FUNCTION_BLOCK FB_LensCompounder_Test EXTENDS TcUnit.FB_TestSuite
VAR
    nTestID : INT;
END_VAR


nTestID := 0;

Test0FocalLengthExpectError0FocalLength();

Test0MultiplierExpectError0FocalLength();

TestNegMultiplierExpectError0FocalLength();

TestResetExpectNoErrorAccurateFocalLength();

TestResetExpectNoErrorAccurateFocalLength_1();

// Expected results taken from pcdscalc/be_lens_calcs.py.
// Element = Be. Test Count = 1.
TestValidInputsExpectNoErrorAccurateFocalLength(
    fFocalLength1 := 0.008893754309452119,
    nMultiplier1 := 1,
    fFocalLength2 := 0.008893754309452119,
    nMultiplier2 := 1,
    fExpected := 0.004446877154726059
);

// Expected results taken from pcdscalc/be_lens_calcs.py.
// Element = Be. Test Count = 2.
TestValidInputsExpectNoErrorAccurateFocalLength(
    fFocalLength1 := 0.008893754309452119,
    nMultiplier1 := 1,
    fFocalLength2 := 0.008893754309452119,
    nMultiplier2 := 2,
    fExpected := 0.002964584769817373
);

// Expected results taken from pcdscalc/be_lens_calcs.py.
// Element = Be. Test Count = 3.
TestValidInputsExpectNoErrorAccurateFocalLength(
    fFocalLength1 := 0.008893754309452119,
    nMultiplier1 := 2,
    fFocalLength2 := 0.008893754309452119,
    nMultiplier2 := 1,
    fExpected := 0.002964584769817373
);

// Expected results taken from pcdscalc/be_lens_calcs.py.
// Element = Be. Test Count = 4.
TestValidInputsExpectNoErrorAccurateFocalLength(
    fFocalLength1 := 0.008893754309452119,
    nMultiplier1 := 2,
    fFocalLength2 := 0.008893754309452119,
    nMultiplier2 := 2,
    fExpected := 0.0022234385773630297
);

// Expected results taken from pcdscalc/be_lens_calcs.py.
// Element = Be. Test Count = 5.
TestValidInputsExpectNoErrorAccurateFocalLength(
    fFocalLength1 := 0.008893754309452119,
    nMultiplier1 := 1,
    fFocalLength2 := 0.45358146978205804,
    nMultiplier2 := 1,
    fExpected := 0.008722720572731886
);

// Expected results taken from pcdscalc/be_lens_calcs.py.
// Element = Be. Test Count = 6.
TestValidInputsExpectNoErrorAccurateFocalLength(
    fFocalLength1 := 0.008893754309452119,
    nMultiplier1 := 1,
    fFocalLength2 := 0.45358146978205804,
    nMultiplier2 := 2,
    fExpected := 0.008558140939284115
);

// Expected results taken from pcdscalc/be_lens_calcs.py.
// Element = Be. Test Count = 7.
TestValidInputsExpectNoErrorAccurateFocalLength(
    fFocalLength1 := 0.008893754309452119,
    nMultiplier1 := 2,
    fFocalLength2 := 0.45358146978205804,
    nMultiplier2 := 1,
    fExpected := 0.004403703590117068
);

// Expected results taken from pcdscalc/be_lens_calcs.py.
// Element = Be. Test Count = 8.
TestValidInputsExpectNoErrorAccurateFocalLength(
    fFocalLength1 := 0.008893754309452119,
    nMultiplier1 := 2,
    fFocalLength2 := 0.45358146978205804,
    nMultiplier2 := 2,
    fExpected := 0.004361360286365943
);

// Expected results taken from pcdscalc/be_lens_calcs.py.
// Element = Be. Test Count = 9.
TestValidInputsExpectNoErrorAccurateFocalLength(
    fFocalLength1 := 0.45358146978205804,
    nMultiplier1 := 1,
    fFocalLength2 := 0.008893754309452119,
    nMultiplier2 := 1,
    fExpected := 0.008722720572731886
);

// Expected results taken from pcdscalc/be_lens_calcs.py.
// Element = Be. Test Count = 10.
TestValidInputsExpectNoErrorAccurateFocalLength(
    fFocalLength1 := 0.45358146978205804,
    nMultiplier1 := 1,
    fFocalLength2 := 0.008893754309452119,
    nMultiplier2 := 2,
    fExpected := 0.004403703590117068
);

// Expected results taken from pcdscalc/be_lens_calcs.py.
// Element = Be. Test Count = 11.
TestValidInputsExpectNoErrorAccurateFocalLength(
    fFocalLength1 := 0.45358146978205804,
    nMultiplier1 := 2,
    fFocalLength2 := 0.008893754309452119,
    nMultiplier2 := 1,
    fExpected := 0.008558140939284115
);

// Expected results taken from pcdscalc/be_lens_calcs.py.
// Element = Be. Test Count = 12.
TestValidInputsExpectNoErrorAccurateFocalLength(
    fFocalLength1 := 0.45358146978205804,
    nMultiplier1 := 2,
    fFocalLength2 := 0.008893754309452119,
    nMultiplier2 := 2,
    fExpected := 0.004361360286365943
);

// Expected results taken from pcdscalc/be_lens_calcs.py.
// Element = Be. Test Count = 13.
TestValidInputsExpectNoErrorAccurateFocalLength(
    fFocalLength1 := 0.45358146978205804,
    nMultiplier1 := 1,
    fFocalLength2 := 0.45358146978205804,
    nMultiplier2 := 1,
    fExpected := 0.22679073489102902
);

// Expected results taken from pcdscalc/be_lens_calcs.py.
// Element = Be. Test Count = 14.
TestValidInputsExpectNoErrorAccurateFocalLength(
    fFocalLength1 := 0.45358146978205804,
    nMultiplier1 := 1,
    fFocalLength2 := 0.45358146978205804,
    nMultiplier2 := 2,
    fExpected := 0.15119382326068603
);

// Expected results taken from pcdscalc/be_lens_calcs.py.
// Element = Be. Test Count = 15.
TestValidInputsExpectNoErrorAccurateFocalLength(
    fFocalLength1 := 0.45358146978205804,
    nMultiplier1 := 2,
    fFocalLength2 := 0.45358146978205804,
    nMultiplier2 := 1,
    fExpected := 0.15119382326068603
);

// Expected results taken from pcdscalc/be_lens_calcs.py.
// Element = Be. Test Count = 16.
TestValidInputsExpectNoErrorAccurateFocalLength(
    fFocalLength1 := 0.45358146978205804,
    nMultiplier1 := 2,
    fFocalLength2 := 0.45358146978205804,
    nMultiplier2 := 2,
    fExpected := 0.11339536744551451
);

// Expected results taken from pcdscalc/be_lens_calcs.py.
// Element = Be. Test Count = 17.
TestValidInputsExpectNoErrorAccurateFocalLength(
    fFocalLength1 := 33.443194804611025,
    nMultiplier1 := 1,
    fFocalLength2 := 33.443194804611025,
    nMultiplier2 := 1,
    fExpected := 16.721597402305513
);

// Expected results taken from pcdscalc/be_lens_calcs.py.
// Element = Be. Test Count = 18.
TestValidInputsExpectNoErrorAccurateFocalLength(
    fFocalLength1 := 33.443194804611025,
    nMultiplier1 := 1,
    fFocalLength2 := 33.443194804611025,
    nMultiplier2 := 2,
    fExpected := 11.147731601537009
);

// Expected results taken from pcdscalc/be_lens_calcs.py.
// Element = Be. Test Count = 19.
TestValidInputsExpectNoErrorAccurateFocalLength(
    fFocalLength1 := 33.443194804611025,
    nMultiplier1 := 2,
    fFocalLength2 := 33.443194804611025,
    nMultiplier2 := 1,
    fExpected := 11.147731601537009
);

// Expected results taken from pcdscalc/be_lens_calcs.py.
// Element = Be. Test Count = 20.
TestValidInputsExpectNoErrorAccurateFocalLength(
    fFocalLength1 := 33.443194804611025,
    nMultiplier1 := 2,
    fFocalLength2 := 33.443194804611025,
    nMultiplier2 := 2,
    fExpected := 8.360798701152756
);

// Expected results taken from pcdscalc/be_lens_calcs.py.
// Element = Be. Test Count = 21.
TestValidInputsExpectNoErrorAccurateFocalLength(
    fFocalLength1 := 33.443194804611025,
    nMultiplier1 := 1,
    fFocalLength2 := 1705.6029350351625,
    nMultiplier2 := 1,
    fExpected := 32.80005644298389
);

// Expected results taken from pcdscalc/be_lens_calcs.py.
// Element = Be. Test Count = 22.
TestValidInputsExpectNoErrorAccurateFocalLength(
    fFocalLength1 := 33.443194804611025,
    nMultiplier1 := 1,
    fFocalLength2 := 1705.6029350351625,
    nMultiplier2 := 2,
    fExpected := 32.18118745349363
);

// Expected results taken from pcdscalc/be_lens_calcs.py.
// Element = Be. Test Count = 23.
TestValidInputsExpectNoErrorAccurateFocalLength(
    fFocalLength1 := 33.443194804611025,
    nMultiplier1 := 2,
    fFocalLength2 := 1705.6029350351625,
    nMultiplier2 := 1,
    fExpected := 16.559251796457886
);

// Expected results taken from pcdscalc/be_lens_calcs.py.
// Element = Be. Test Count = 24.
TestValidInputsExpectNoErrorAccurateFocalLength(
    fFocalLength1 := 33.443194804611025,
    nMultiplier1 := 2,
    fFocalLength2 := 1705.6029350351625,
    nMultiplier2 := 2,
    fExpected := 16.400028221491944
);

// Expected results taken from pcdscalc/be_lens_calcs.py.
// Element = Be. Test Count = 25.
TestValidInputsExpectNoErrorAccurateFocalLength(
    fFocalLength1 := 1705.6029350351625,
    nMultiplier1 := 1,
    fFocalLength2 := 33.443194804611025,
    nMultiplier2 := 1,
    fExpected := 32.80005644298389
);

// Expected results taken from pcdscalc/be_lens_calcs.py.
// Element = Be. Test Count = 26.
TestValidInputsExpectNoErrorAccurateFocalLength(
    fFocalLength1 := 1705.6029350351625,
    nMultiplier1 := 1,
    fFocalLength2 := 33.443194804611025,
    nMultiplier2 := 2,
    fExpected := 16.559251796457886
);

// Expected results taken from pcdscalc/be_lens_calcs.py.
// Element = Be. Test Count = 27.
TestValidInputsExpectNoErrorAccurateFocalLength(
    fFocalLength1 := 1705.6029350351625,
    nMultiplier1 := 2,
    fFocalLength2 := 33.443194804611025,
    nMultiplier2 := 1,
    fExpected := 32.18118745349363
);

// Expected results taken from pcdscalc/be_lens_calcs.py.
// Element = Be. Test Count = 28.
TestValidInputsExpectNoErrorAccurateFocalLength(
    fFocalLength1 := 1705.6029350351625,
    nMultiplier1 := 2,
    fFocalLength2 := 33.443194804611025,
    nMultiplier2 := 2,
    fExpected := 16.400028221491944
);

// Expected results taken from pcdscalc/be_lens_calcs.py.
// Element = Be. Test Count = 29.
TestValidInputsExpectNoErrorAccurateFocalLength(
    fFocalLength1 := 1705.6029350351625,
    nMultiplier1 := 1,
    fFocalLength2 := 1705.6029350351625,
    nMultiplier2 := 1,
    fExpected := 852.8014675175812
);

// Expected results taken from pcdscalc/be_lens_calcs.py.
// Element = Be. Test Count = 30.
TestValidInputsExpectNoErrorAccurateFocalLength(
    fFocalLength1 := 1705.6029350351625,
    nMultiplier1 := 1,
    fFocalLength2 := 1705.6029350351625,
    nMultiplier2 := 2,
    fExpected := 568.5343116783874
);

// Expected results taken from pcdscalc/be_lens_calcs.py.
// Element = Be. Test Count = 31.
TestValidInputsExpectNoErrorAccurateFocalLength(
    fFocalLength1 := 1705.6029350351625,
    nMultiplier1 := 2,
    fFocalLength2 := 1705.6029350351625,
    nMultiplier2 := 1,
    fExpected := 568.5343116783874
);

// Expected results taken from pcdscalc/be_lens_calcs.py.
// Element = Be. Test Count = 32.
TestValidInputsExpectNoErrorAccurateFocalLength(
    fFocalLength1 := 1705.6029350351625,
    nMultiplier1 := 2,
    fFocalLength2 := 1705.6029350351625,
    nMultiplier2 := 2,
    fExpected := 426.4007337587906
);


METHOD Test0FocalLengthExpectError0FocalLength
VAR
    // Subject under test
    fbLensCompounder : FB_LensCompounder();
END_VAR

TEST('Test0FocalLengthExpectError0FocalLength');

// Test fixture
fbLensCompounder.Reset();

// Here the test starts
fbLensCompounder.Compound(
    fFocalLength := 0.0,
    nMultiplier := 1
);

AssertTrue(
    Condition := fbLensCompounder.GetError(),
    Message := 'Expected bError bit to be true but it was false.'
);

AssertTrue(
    Condition := fbLensCompounder.GetErrorMsg() <> '',
    Message := 'Expected sErrorMsg to not be empty.'
);

AssertEquals_LREAL(
    Expected := 0,
    Actual := fbLensCompounder.FocalLengthCompounded,
    Delta := 0,
    Message := 'Calculated focal length compounded should be 0 when an error is detected.'
);

TEST_FINISHED();
END_METHOD


METHOD Test0MultiplierExpectError0FocalLength
VAR
    // Subject under test
    fbLensCompounder : FB_LensCompounder();
END_VAR

TEST('Test0MultiplierExpectError0FocalLength');

// Test fixture
fbLensCompounder.Reset();

// Here the test starts
fbLensCompounder.Compound(
    fFocalLength := 1.0,
    nMultiplier := 0
);

AssertTrue(
    Condition := fbLensCompounder.GetError(),
    Message := 'Expected bError bit to be true but it was false.'
);

AssertTrue(
    Condition := fbLensCompounder.GetErrorMsg() <> '',
    Message := 'Expected sErrorMsg to not be empty.'
);

AssertEquals_LREAL(
    Expected := 0,
    Actual := fbLensCompounder.FocalLengthCompounded,
    Delta := 0,
    Message := 'Calculated focal length compounded should be 0 when an error is detected.'
);

TEST_FINISHED();
END_METHOD


METHOD TestNegMultiplierExpectError0FocalLength
VAR
    // Subject under test
    fbLensCompounder : FB_LensCompounder();
END_VAR

TEST('TestNegMultiplierExpectError0FocalLength');

// Test fixture
fbLensCompounder.Reset();

// Here the test starts
fbLensCompounder.Compound(
    fFocalLength := 1.0,
    nMultiplier := -1
);

AssertTrue(
    Condition := fbLensCompounder.GetError(),
    Message := 'Expected bError bit to be true but it was false.'
);

AssertTrue(
    Condition := fbLensCompounder.GetErrorMsg() <> '',
    Message := 'Expected sErrorMsg to not be empty.'
);

AssertEquals_LREAL(
    Expected := 0,
    Actual := fbLensCompounder.FocalLengthCompounded,
    Delta := 0,
    Message := 'Calculated focal length compounded should be 0 when an error is detected.'
);

TEST_FINISHED();
END_METHOD


METHOD TestResetExpectNoErrorAccurateFocalLength
VAR
    // Subject under test
    fbLensCompounder : FB_LensCompounder();
END_VAR

TEST('TestResetExpectNoErrorAccurateFocalLength');

// Test fixture
fbLensCompounder.Reset();

// Here the test starts
fbLensCompounder.Compound(
    fFocalLength := 1.0,
    nMultiplier := 1
);

fbLensCompounder.Reset();

AssertFalse(
    Condition := fbLensCompounder.GetError(),
    Message := 'Expected bError bit to be false but it was true.'
);

AssertFalse(
    Condition := fbLensCompounder.GetErrorMsg() <> '',
    Message := 'Expected sErrorMsg to be empty.'
);

AssertEquals_LREAL(
    Expected := 0.0,
    Actual := fbLensCompounder.FocalLengthCompounded,
    Delta := 0.0,
    Message := 'Calculated focal length did not calculate close enough to the expected value.'
);

TEST_FINISHED();

nTestID := nTestID + 1;
END_METHOD


METHOD TestResetExpectNoErrorAccurateFocalLength_1
VAR
    // Subject under test
    fbLensCompounder : FB_LensCompounder();
END_VAR

TEST('TestResetExpectNoErrorAccurateFocalLength_1');

// Test fixture
fbLensCompounder.Reset();

// Here the test starts
fbLensCompounder.Compound(
    fFocalLength := 1.0,
    nMultiplier := 1
);

fbLensCompounder.Reset();

fbLensCompounder.Compound(
    fFocalLength := 1.0,
    nMultiplier := 1
);

AssertFalse(
    Condition := fbLensCompounder.GetError(),
    Message := 'Expected bError bit to be false but it was true.'
);

AssertFalse(
    Condition := fbLensCompounder.GetErrorMsg() <> '',
    Message := 'Expected sErrorMsg to be empty.'
);

AssertEquals_LREAL(
    Expected := 1.0,
    Actual := fbLensCompounder.FocalLengthCompounded,
    Delta := 1.0,
    Message := 'Calculated focal length did not calculate close enough to the expected value.'
);

TEST_FINISHED();

nTestID := nTestID + 1;
END_METHOD


METHOD TestValidInputsExpectNoErrorAccurateFocalLength
VAR_INPUT
    fFocalLength1 : LREAL;
    nMultiplier1 : INT;
    fFocalLength2 : LREAL;
    nMultiplier2 : INT;

    fExpected : LREAL;
END_VAR
VAR
    // Subject under test
    fbLensCompounder : FB_LensCompounder();
END_VAR

TEST(CONCAT(STR1 := 'TestValidInputsExpectNoErrorAccurateFocalLength ID: ',
            STR2 := INT_TO_STRING(nTestID)));

// Test fixture
fbLensCompounder.Reset();

// Here the test starts
fbLensCompounder.Compound(
    fFocalLength := fFocalLength1,
    nMultiplier := nMultiplier1
);

fbLensCompounder.Compound(
    fFocalLength := fFocalLength2,
    nMultiplier := nMultiplier2
);

AssertFalse(
    Condition := fbLensCompounder.GetError(),
    Message := 'Expected bError bit to be false but it was true.'
);

AssertFalse(
    Condition := fbLensCompounder.GetErrorMsg() <> '',
    Message := 'Expected sErrorMsg to be empty.'
);

AssertEquals_LREAL(
    Expected := fExpected,
    Actual := fbLensCompounder.FocalLengthCompounded,
    Delta := ABS(0.001 * fExpected),
    Message := 'Calculated focal length did not calculate close enough to the expected value.'
);

TEST_FINISHED();

nTestID := nTestID + 1;
END_METHOD

END_FUNCTION_BLOCK

(* stored: Version 1.1.0.1
   POU FB_LensCompounder_Test: Id {f7d35265-95ed-426e-abbf-8e10febba493}, SpecialFunc None
   Method Test0FocalLengthExpectError0FocalLength: Id {b281f112-8ce2-43a7-9e96-9df05b42c757}
   Method Test0MultiplierExpectError0FocalLength: Id {07524415-12aa-410c-946c-4f8ae36284dd}
   Method TestNegMultiplierExpectError0FocalLength: Id {0a50e7fc-0cd1-4e4a-bc10-32e5185f3a93}
   Method TestResetExpectNoErrorAccurateFocalLength: Id {076846fa-8184-45ab-be3a-11c83773551f}
   Method TestResetExpectNoErrorAccurateFocalLength_1: Id {d8699e2c-b50f-4b10-b5ff-eadd751cdc81}
   Method TestValidInputsExpectNoErrorAccurateFocalLength: Id {ebe91652-846f-46fc-946b-f0c6b61f529d} *)
